# B&R Automation Studio project SceneViewer
Automation Studio 4.7.3.93 SP; technology packages: mappMotion 5.13.1, mappView 5.13.0

## Configuration Config1

CPU PC_any, AutomationRuntime B4.73, Build 4.1.2, Safety 0.0, Vc V4.72.3

### Task classes (Cpu.sw)
```
Cyclic#1 (cycle 1000 us, tolerance 0 us):
  Vis <- Vis.prg
  Trak <- Trak.prg
  SVControl <- SVControl.prg
DataObjects: McAcpSys
Binaries: FWRules, McAcpSim, arcoal, arsvcreg, TCData, McAcpDrv, arflatprv, udbdef, mvLoader, iomap, Config_1, arconfig, asfw, ashwac, sysconf, User, Role, ashwd, Config_3
Libraries: BeEasyTrak, SceneView, McBase, McAxis, McAcpTrak, standard, AsBrStr, AsMath, MpAxis, MpBase, McAcpAx, runtime, astime, fileio, powerlnk, asieccon, arssl
```

### Hardware
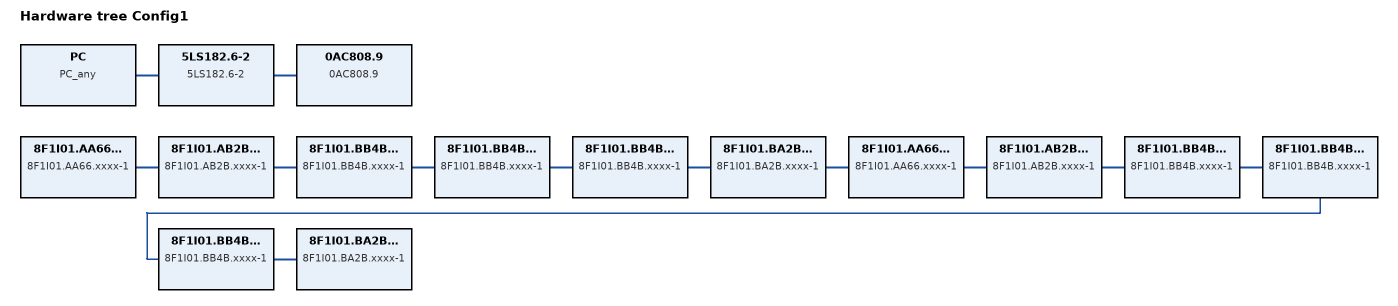
```
0AC808.9 : 0AC808.9 v1.0.0.0  [ETH1 -> 5LS182.6-2.IF1 [Cable Type=PowerlinkCable, Length=10, Version=1.0.0.2]; ETH2 -> 8F1I01.AA66.xxxx-1.PLK3 [Cable Type=PowerlinkCable, Length=10, Version=1.0.0.2]]
5LS182.6-2 : 5LS182.6-2 v1.7.0.0  [SL -> PC.SL1]
8F1I01.AA66.xxxx-1 : 8F1I01.AA66.xxxx-1 v1.0.0.2  [PLK2 -> 8F1I01.AB2B.xxxx-1.PLK1 [Cable Type=PowerlinkCable, Length=10, Version=1.0.0.2]; PLK3 -> 0AC808.9.ETH2 [Cable Type=PowerlinkCable, Length=10, Version=1.0.0.2]]
  DriveConfiguration:
    McTypeID = LLMConfig
  DriveConfiguration/Segment:
    Shape = STRAIGHT660
    SegmentReference = gSeg_Main_1
    StopReaction = UseAssemblySetting
    SpeedFilter = UseAssemblySetting
8F1I01.AA66.xxxx-1a : 8F1I01.AA66.xxxx-1 v1.0.0.2  [PLK1 -> 8F1I01.BA2B.xxxx-1a.PLK2 [Cable Type=PowerlinkCable, Length=10, Version=1.0.0.2]; PLK2 -> 8F1I01.AB2B.xxxx-1a.PLK1 [Cable Type=PowerlinkCable, Length=10, Version=1.0.0.2]]
  DriveConfiguration:
    McTypeID = LLMConfig
  DriveConfiguration/Segment:
    Shape = STRAIGHT660
    SegmentReference = gSeg_Main_7
    StopReaction = UseAssemblySetting
    SpeedFilter = UseAssemblySetting
8F1I01.AB2B.xxxx-1 : 8F1I01.AB2B.xxxx-1 v1.0.0.2  [PLK1 -> 8F1I01.AA66.xxxx-1.PLK2 [Cable Type=PowerlinkCable, Length=10, Version=1.0.0.2]; PLK2 -> 8F1I01.BB4B.xxxx-1.PLK1 [Cable Type=PowerlinkCable, Length=10, Version=1.0.0.2]]
  DriveConfiguration:
    McTypeID = LLMConfig
  DriveConfiguration/Segment:
    Shape = STRAIGHT105_TO_CIRCULAR
    SegmentReference = gSeg_Main_2
    StopReaction = UseAssemblySetting
    SpeedFilter = UseAssemblySetting
8F1I01.AB2B.xxxx-1a : 8F1I01.AB2B.xxxx-1 v1.0.0.2  [PLK1 -> 8F1I01.AA66.xxxx-1a.PLK2 [Cable Type=PowerlinkCable, Length=10, Version=1.0.0.2]; PLK2 -> 8F1I01.BB4B.xxxx-1c.PLK1 [Cable Type=PowerlinkCable, Length=10, Version=1.0.0.2]]
  DriveConfiguration:
    McTypeID = LLMConfig
  DriveConfiguration/Segment:
    Shape = STRAIGHT105_TO_CIRCULAR
    SegmentReference = gSeg_Main_8
    StopReaction = UseAssemblySetting
    SpeedFilter = UseAssemblySetting
8F1I01.BA2B.xxxx-1 : 8F1I01.BA2B.xxxx-1 v1.0.0.2  [PLK1 -> 8F1I01.BB4B.xxxx-1e.PLK2 [Cable Type=PowerlinkCable, Length=10, Version=1.0.0.2]]
  DriveConfiguration:
    McTypeID = LLMConfig
  DriveConfiguration/Segment:
    Shape = CIRCULAR_TO_STRAIGHT105
    SegmentReference = gSeg_Main_12
    StopReaction = UseAssemblySetting
    SpeedFilter = UseAssemblySetting
8F1I01.BA2B.xxxx-1a : 8F1I01.BA2B.xxxx-1 v1.0.0.2  [PLK1 -> 8F1I01.BB4B.xxxx-1b.PLK2 [Cable Type=PowerlinkCable, Length=10, Version=1.0.0.2]; PLK2 -> 8F1I01.AA66.xxxx-1a.PLK1 [Cable Type=PowerlinkCable, Length=10, Version=1.0.0.2]]
  DriveConfiguration:
    McTypeID = LLMConfig
  DriveConfiguration/Segment:
    Shape = CIRCULAR_TO_STRAIGHT105
    SegmentReference = gSeg_Main_6
    StopReaction = UseAssemblySetting
    SpeedFilter = UseAssemblySetting
8F1I01.BB4B.xxxx-1 : 8F1I01.BB4B.xxxx-1 v1.0.0.2  [PLK1 -> 8F1I01.AB2B.xxxx-1.PLK2 [Cable Type=PowerlinkCable, Length=10, Version=1.0.0.2]; PLK2 -> 8F1I01.BB4B.xxxx-1a.PLK1 [Cable Type=PowerlinkCable, Length=10, Version=1.0.0.2]]
  DriveConfiguration:
    McTypeID = LLMConfig
  DriveConfiguration/Segment:
    Shape = CIRCULAR
    SegmentReference = gSeg_Main_3
    StopReaction = UseAssemblySetting
    SpeedFilter = UseAssemblySetting
8F1I01.BB4B.xxxx-1a : 8F1I01.BB4B.xxxx-1 v1.0.0.2  [PLK1 -> 8F1I01.BB4B.xxxx-1.PLK2 [Cable Type=PowerlinkCable, Length=10, Version=1.0.0.2]; PLK2 -> 8F1I01.BB4B.xxxx-1b.PLK1 [Cable Type=PowerlinkCable, Length=10, Version=1.0.0.2]]
  DriveConfiguration:
    McTypeID = LLMConfig
  DriveConfiguration/Segment:
    Shape = CIRCULAR
    SegmentReference = gSeg_Main_4
    StopReaction = UseAssemblySetting
    SpeedFilter = UseAssemblySetting
8F1I01.BB4B.xxxx-1b : 8F1I01.BB4B.xxxx-1 v1.0.0.2  [PLK1 -> 8F1I01.BB4B.xxxx-1a.PLK2 [Cable Type=PowerlinkCable, Length=10, Version=1.0.0.2]; PLK2 -> 8F1I01.BA2B.xxxx-1a.PLK1 [Cable Type=PowerlinkCable, Length=10, Version=1.0.0.2]]
  DriveConfiguration:
    McTypeID = LLMConfig
  DriveConfiguration/Segment:
    Shape = CIRCULAR
    SegmentReference = gSeg_Main_5
    StopReaction = UseAssemblySetting
    SpeedFilter = UseAssemblySetting
8F1I01.BB4B.xxxx-1c : 8F1I01.BB4B.xxxx-1 v1.0.0.2  [PLK1 -> 8F1I01.AB2B.xxxx-1a.PLK2 [Cable Type=PowerlinkCable, Length=10, Version=1.0.0.2]; PLK2 -> 8F1I01.BB4B.xxxx-1d.PLK1 [Cable Type=PowerlinkCable, Length=10, Version=1.0.0.2]]
  DriveConfiguration:
    McTypeID = LLMConfig
  DriveConfiguration/Segment:
    Shape = CIRCULAR
    SegmentReference = gSeg_Main_9
    StopReaction = UseAssemblySetting
    SpeedFilter = UseAssemblySetting
8F1I01.BB4B.xxxx-1d : 8F1I01.BB4B.xxxx-1 v1.0.0.2  [PLK1 -> 8F1I01.BB4B.xxxx-1c.PLK2 [Cable Type=PowerlinkCable, Length=10, Version=1.0.0.2]; PLK2 -> 8F1I01.BB4B.xxxx-1e.PLK1 [Cable Type=PowerlinkCable, Length=10, Version=1.0.0.2]]
  DriveConfiguration:
    McTypeID = LLMConfig
  DriveConfiguration/Segment:
    Shape = CIRCULAR
    SegmentReference = gSeg_Main_10
    StopReaction = UseAssemblySetting
    SpeedFilter = UseAssemblySetting
8F1I01.BB4B.xxxx-1e : 8F1I01.BB4B.xxxx-1 v1.0.0.2  [PLK1 -> 8F1I01.BB4B.xxxx-1d.PLK2 [Cable Type=PowerlinkCable, Length=10, Version=1.0.0.2]; PLK2 -> 8F1I01.BA2B.xxxx-1.PLK1 [Cable Type=PowerlinkCable, Length=10, Version=1.0.0.2]]
  DriveConfiguration:
    McTypeID = LLMConfig
  DriveConfiguration/Segment:
    Shape = CIRCULAR
    SegmentReference = gSeg_Main_11
    StopReaction = UseAssemblySetting
    SpeedFilter = UseAssemblySetting
PC : PC_any v1.1.0.0 (OrderNumber=PC)
  ConfigurationID = SceneViewer_Config1
  SystemTick = 1000
  Cyclic1Duration = 1000
  Cyclic1Tolerance = 0
  Cyclic2Duration = 2000
  FileDevice1
  FileDeviceName1 = SvgData
  FileDevicePath1 = C:\Trak\Scene
  ActivateOpcUa = 1
  OpcUaInformationModels_PV_Version = 1
```

### Config_1.assembly - PC/mappMotion/Config_1.assembly
```
Element gAssembly_1 (Type=assembly)
  Tracks:
    TrackSeparation = 0.030
    Track[1]:
      Segments:
        SegmentRef[1] = ::gSeg_Main_1
        SegmentRef[2] = ::gSeg_Main_2
        SegmentRef[3] = ::gSeg_Main_3
        SegmentRef[4] = ::gSeg_Main_4
        SegmentRef[5] = ::gSeg_Main_5
        SegmentRef[6] = ::gSeg_Main_6
        SegmentRef[7] = ::gSeg_Main_7
        SegmentRef[8] = ::gSeg_Main_8
        SegmentRef[9] = ::gSeg_Main_9
        SegmentRef[10] = ::gSeg_Main_10
        SegmentRef[11] = ::gSeg_Main_11
        SegmentRef[12] = ::gSeg_Main_12
      Position = Absolute
        SegmentCountDirection = RightToLeft
        Translation:
          X = 0.0
          Y = 0.0
          Z = 0.0
        Orientation:
          Angle1 = 0.0
          Angle2 = 0.0
          Angle3 = 0.0
  CommonSegmentSettings:
    SegmentSimulationOnPLC = Off
    StopReaction = InductionHalt
    SpeedFilter = NotUsed
    ControllerParameters:
      DefaultParameter:
        Controller:
          Position:
            ProportionalGain = 0.0
          Speed:
            ProportionalGain = 0.0
            IntegrationTime = 0.0
          FeedForward:
            TotalMass = 0.0
            ForcePositive = 0.0
            ForceNegative = 0.0
            SpeedForceFactor = 0.0
            ForceLoad = 0.0
        MovementErrorLimits:
          PositionError = 0.0
          VelocityError = 0.0
      AdditionalParameterSets = NotUsed
    ScopeOfErrorReaction = Assembly
    ShuttleIdentificationTime = 0
  Shuttles:
    MaxShuttleCount = 10
    DistanceReserve:
      Collision = 0.002
      ErrorStop = 0.006
    ShuttleStereotypes:
      ShuttleStRef[1] = ShuttleStereotype_1
    MagnetPlateConfigurations:
      ShuttleType[1] = 8F1SA.100.xxxxxx-x
    CollisionAvoidance:
      Strategy = Constant
      MaximumModelDimensions:
        Length:
          ExtentToFront = 0.025
          ExtentToBack = 0.025
        Width:
          Width = 0.046
  AssemblyFeatures:
    AssemblyFeatureRef[1] = AssemblyFeature_1
  Visualization:
    MonitoringPv = ::gShuttleMon
    ProcessingTaskClass = 2
```

### Config_2.sector - PC/mappMotion/Config_2.sector
```
Element Sector_1 (Type=sector)
  Type = Composed
    StartSegment:
      SegmentRef = ::gSeg_Main_1
    IntermediateSegments:
      SegmentRef[1] = ::gSeg_Main_2
      SegmentRef[2] = ::gSeg_Main_3
      SegmentRef[3] = ::gSeg_Main_4
      SegmentRef[4] = ::gSeg_Main_5
      SegmentRef[5] = ::gSeg_Main_6
      SegmentRef[6] = ::gSeg_Main_7
      SegmentRef[7] = ::gSeg_Main_8
      SegmentRef[8] = ::gSeg_Main_9
      SegmentRef[9] = ::gSeg_Main_10
      SegmentRef[10] = ::gSeg_Main_11
    EndSegment:
      SegmentRef = ::gSeg_Main_12
      PositionRelativeTo = FromEnd
```

### Config_3.shuttlestereotype - PC/mappMotion/Config_3.shuttlestereotype
```
Element ShuttleStereotype_1 (Type=shuttlestereotype)
  MeasurementUnit = 5067858
  MeasurementResolution = 0.00001
  MovementLimits = Internal
    VelocityIsReadOnly = 0
    Velocity:
      Velocity = 4.0
    AccelerationIsReadOnly = 0
    Acceleration:
      Acceleration = 20
    DecelerationIsReadOnly = 0
    Deceleration:
      Deceleration = 20
  JerkFilter = Used
    JerkTime = 0.02
  UserData:
    Size = 0
```

### Config_4.assemblyfeature - PC/mappMotion/Config_4.assemblyfeature
```
Element AssemblyFeature_1 (Type=assemblyfeature)
  Type = InitShuttleSim
    InitShuttleSim[1]:
      SectorRef = Sector_1
      Orientation = Positive
      ShuttleDefinition = ShuttleSetDefinition
        StartPosition = 0.0
        NumberOfShuttles = 5
        DistnaceBetweenShuttles = 0.2
```

### cfgSV.mprecipexml - PC/mappServices/cfgSV.mprecipexml
```
Element gRecipeScnViewer (Type=mprecipexml)
```

## Logical view

Binary libraries used (declarations not repeated): operator, runtime, astime, AsIecCon, McBase 5.13.1, McAxis 5.13.1, McAcpTrak 5.13.1, standard, AsBrStr, AsMath, MpAxis 5.13.1, MpBase 5.13.0, McAcpAx 5.13.1

### Segments.var
```iecst
VAR
	gSeg_Main_1 : McSegmentType;
	gSeg_Main_2 : McSegmentType;
	gSeg_Main_3 : McSegmentType;
	gSeg_Main_4 : McSegmentType;
	gSeg_Main_5 : McSegmentType;
	gSeg_Main_6 : McSegmentType;
	gSeg_Main_7 : McSegmentType;
	gSeg_Main_8 : McSegmentType;
	gSeg_Main_9 : McSegmentType;
	gSeg_Main_10 : McSegmentType;
	gSeg_Main_11 : McSegmentType;
	gSeg_Main_12 : McSegmentType;
END_VAR
```

### Package Logical/Libraries - Global libraries

### Library Logical/Libraries/BeEasyTrak (IEC)

#### Types.typ - Exported data types
```iecst
TYPE
	Barrier_typ : 	STRUCT
		BarrierReadInfo : MC_BR_BarrierReadInfo_AcpTrak;
		BarrierCommand : MC_BR_BarrierCommand_AcpTrak;
	END_STRUCT;
	TrgPoint_typ : 	STRUCT
		TrgPointGetInfo : MC_BR_TrgPointGetInfo_AcpTrak;
		TrgPointEnable : MC_BR_TrgPointEnable_AcpTrak;
	END_STRUCT;
	ShuttleUserData_typ : 	STRUCT
		Color : Color_enum;
	END_STRUCT;
	Color_enum :
		(
		GRAY := 0,
		GREEN := 1,
		BLUE := 2,
		RED := 3,
		ORANGE := 4,
		YELLOW,
		WHITE
		);
END_TYPE
```

#### Constants.var - Exported constants
```iecst
VAR CONSTANT
	MAX_SHUTTLES : UINT := 5;
	NUM_SHUTTLES : UINT := 5;
END_VAR
```

#### BeEasyTrak.fun - Exported functions and function blocks
```iecst
{REDUND_ERROR} FUNCTION_BLOCK BE_TrgPoint (*TODO: Add your comment here*) (*$GROUP=User,$CAT=User,$GROUPICON=User.png,$CATICON=User.png*)
	VAR_INPUT
		ProcessPoint : REFERENCE TO McProcessPointType;
		Enable : BOOL;
	END_VAR
	VAR_OUTPUT
		ShuttleAxis : McAxisType;
		Triggered : BOOL;
	END_VAR
	VAR
		State : USINT;
		TrgPoint : TrgPoint_typ;
	END_VAR
END_FUNCTION_BLOCK

{REDUND_ERROR} FUNCTION_BLOCK BE_SimStartup (*TODO: Add your comment here*) (*$GROUP=User,$CAT=User,$GROUPICON=User.png,$CATICON=User.png*)
	VAR_INPUT
		Assembly : REFERENCE TO McAssemblyType;
		Sector : REFERENCE TO McSectorType;
		Execute : BOOL;
	END_VAR
	VAR_OUTPUT
		ShuttleAxisArray : ARRAY[1..MAX_SHUTTLES] OF McAxisType;
		Done : BOOL;
	END_VAR
	VAR
		AsmReadInfo : MC_BR_AsmReadInfo_AcpTrak;
		AddShuttle : MC_BR_SecAddShuttle_AcpTrak;
		ElasticMoveVel : MC_BR_ElasticMoveVel_AcpTrak;
		State : USINT;
		i : USINT := 1;
		zzEdge00000 : BOOL;
	END_VAR
END_FUNCTION_BLOCK

{REDUND_ERROR} FUNCTION_BLOCK BE_Rate (*TODO: Add your comment here*) (*$GROUP=User,$CAT=User,$GROUPICON=User.png,$CATICON=User.png*)
	VAR_INPUT
		ProcessPoint : REFERENCE TO McProcessPointType;
		Enable : BOOL;
	END_VAR
	VAR_OUTPUT
		PPM : UINT;
		PPM_Instant : REAL;
		PPH : UINT;
		PPH_Instant : REAL;
	END_VAR
	VAR
		Counter : UINT;
		State : USINT;
		TrgPoint : BE_TrgPoint;
		TON_InstantRate : TON;
		TON_PPM : TON;
	END_VAR
END_FUNCTION_BLOCK

{REDUND_ERROR} FUNCTION_BLOCK BE_FindShuttles (*TODO: Add your comment here*) (*$GROUP=User,$CAT=User,$GROUPICON=User.png,$CATICON=User.png*)
	VAR_INPUT
		Assembly : REFERENCE TO USINT;
		Execute : {REDUND_UNREPLICABLE} BOOL;
	END_VAR
	VAR_OUTPUT
		NumShuttlesFound : UINT;
		ShuttleAxisArray : ARRAY[1..MAX_SHUTTLES] OF McAxisType;
		Done : {REDUND_UNREPLICABLE} BOOL;
		Error : BOOL;
		Busy : BOOL;
	END_VAR
	VAR
		i : USINT;
		AsmGetShuttle : MC_BR_AsmGetShuttle_AcpTrak;
		State : USINT;
	END_VAR
END_FUNCTION_BLOCK

{REDUND_ERROR} FUNCTION_BLOCK BE_MoveOnSector (*TODO: Add your comment here*) (*$GROUP=User,$CAT=User,$GROUPICON=User.png,$CATICON=User.png*)
	VAR_INPUT
		Execute : {REDUND_UNREPLICABLE} BOOL;
		Sector : REFERENCE TO McSectorType;
		Velocity : REAL;
		Acceleration : REAL;
		Deceleration : REAL;
		AxisArray : ARRAY[1..MAX_SHUTTLES] OF McAxisType;
		Assembly : REFERENCE TO McAssemblyType;
	END_VAR
	VAR_OUTPUT
		NumShuttles : UINT;
		Done : {REDUND_UNREPLICABLE} BOOL;
	END_VAR
	VAR
		RoutedMoveVel : MC_BR_RoutedMoveVel_AcpTrak;
		AsmGetShuttle : MC_BR_AsmGetShuttle_AcpTrak;
		i : UINT;
		State : USINT;
		zzEdge00000 : BOOL;
	END_VAR
END_FUNCTION_BLOCK

{REDUND_ERROR} FUNCTION_BLOCK BE_AsmStop (*TODO: Add your comment here*) (*$GROUP=User,$CAT=User,$GROUPICON=User.png,$CATICON=User.png*)
	VAR_INPUT
		Execute : {REDUND_UNREPLICABLE} BOOL;
		AxisArray : {REDUND_UNREPLICABLE} ARRAY[1..MAX_SHUTTLES] OF McAxisType;
		Deceleration : REAL;
		NumShuttles : UINT;
	END_VAR
	VAR_OUTPUT
		Done : {REDUND_UNREPLICABLE} BOOL;
	END_VAR
	VAR
		State : USINT;
		Stop : MC_Stop;
		i : UINT;
	END_VAR
END_FUNCTION_BLOCK
```

#### BE_TrgPoint.st
```iecst
(* TODO: Add your comment here *)
FUNCTION_BLOCK BE_TrgPoint

	TrgPoint.TrgPointEnable.ProcessPoint := ADR(ProcessPoint);
	TrgPoint.TrgPointGetInfo.ProcessPoint := ADR(ProcessPoint);

	TrgPoint.TrgPointEnable.Enable := Enable;

	CASE State OF
		0:
			IF TrgPoint.TrgPointEnable.EventCount > 0 THEN
				TrgPoint.TrgPointGetInfo.Execute := TRUE;
			END_IF

			IF TrgPoint.TrgPointGetInfo.TrgPointInfo.Event = mcACPTRAK_TP_PASSED_POSITIVE THEN
				ShuttleAxis := TrgPoint.TrgPointGetInfo.TrgPointInfo.Axis;
				TrgPoint.TrgPointGetInfo.Execute := FALSE;
				Triggered := TRUE;
				State := 1;
			END_IF

		1:
			Triggered := FALSE;
			State := 0;

	END_CASE

	TrgPoint.TrgPointEnable();
	TrgPoint.TrgPointGetInfo();

END_FUNCTION_BLOCK
```

#### BE_SimStartup.st
```iecst
(* TODO: Add your comment here *)
FUNCTION_BLOCK BE_SimStartup

	AsmReadInfo.Assembly := ADR(Assembly);
	AsmReadInfo.Enable := TRUE;

	CASE State OF
		0: //POWER_ON
			IF Execute THEN
				State := 1;
			END_IF

		1: //ADD_SHUTTLES
			AddShuttle.Sector := ADR(Sector);
			AddShuttle.Position := (i - 1) * 0.1;
			AddShuttle.Execute := TRUE;

			IF AddShuttle.Done  THEN
				ShuttleAxisArray[i] := AddShuttle.Axis;
				AddShuttle.Execute := FALSE;
				i := i + 1;
			END_IF

			IF i > NUM_SHUTTLES THEN
				i := 1;
				State := 2;
			END_IF

		2: //MOVE_SHUTTLES

			IF EDGEPOS(ElasticMoveVel.Active) THEN
				i := i + 1;
			ELSIF ShuttleAxisArray[i].controlif <> 0 THEN
				ElasticMoveVel.Axis := ADR(ShuttleAxisArray[i]);
				ElasticMoveVel.Velocity := 2;
				ElasticMoveVel.Acceleration := 10;
				ElasticMoveVel.Deceleration := 10;
				ElasticMoveVel.Execute := TRUE;
			END_IF

			IF i > NUM_SHUTTLES THEN
				State := 3;
			END_IF
//
		3: //STANDBY
			Done := TRUE;
			IF NOT Execute THEN
				Done := FALSE;
				State := 0;
			END_IF

	END_CASE

	AddShuttle();
	AsmReadInfo();
	ElasticMoveVel();
	ElasticMoveVel.Execute := FALSE;

END_FUNCTION_BLOCK
```

#### BE_Rate.st
```iecst
(* TODO: Add your comment here *)
FUNCTION_BLOCK BE_Rate

	CASE State OF
		0:
			IF Enable THEN
				State := 1;
			END_IF

		1:
			TON_InstantRate.PT := T#60m;
			TON_InstantRate.IN := TRUE;

			TrgPoint.ProcessPoint := ADR(ProcessPoint);
			TrgPoint.Enable := TRUE;

			IF TrgPoint.Triggered THEN
				Counter := Counter + 1;

				TON_InstantRate.IN := FALSE;
				IF TIME_TO_REAL(TON_InstantRate.ET) <> 0 THEN
					PPM_Instant := 1000 / TIME_TO_REAL(TON_InstantRate.ET);
					PPH_Instant := 60 * 1000 / TIME_TO_REAL(TON_InstantRate.ET);
				END_IF
			END_IF

			TON_PPM.PT := T#60s;
			TON_PPM.IN := TRUE;

			IF TON_PPM.Q THEN
				TON_PPM.IN := FALSE;
				PPM := Counter;
				Counter := 0;
			END_IF

			PPH := PPM * 60;

	END_CASE

	TON_InstantRate;
	TrgPoint();
	TON_PPM();

END_FUNCTION_BLOCK
```

#### BE_FindShuttles.st
```iecst
(* TODO: Add your comment here *)
FUNCTION_BLOCK BE_FindShuttles
	AsmGetShuttle.Assembly := ADR(Assembly);

	IF AsmGetShuttle.Error THEN
		Error := TRUE;
		State := 4;
	END_IF

	CASE State OF
		0:
			IF Execute THEN
				i := 1;
				Busy := TRUE;
				State := 1;
			END_IF

		1:
			AsmGetShuttle.Enable := TRUE;
			IF AsmGetShuttle.Valid THEN
				NumShuttlesFound := AsmGetShuttle.TotalCount;
				IF AsmGetShuttle.Axis.controlif <> 0 THEN
					ShuttleAxisArray[i] := AsmGetShuttle.Axis;
				END_IF
				IF AsmGetShuttle.RemainingCount > 0 THEN
					AsmGetShuttle.Next := TRUE;
					State := 2;
				ELSE
					State := 3;
				END_IF
			END_IF

		2:
			AsmGetShuttle.Next := FALSE;
			i := i + 1;
			State := 1;

		3:
			Done := TRUE;
			IF NOT Execute THEN
				brsmemset(ADR(ShuttleAxisArray),0,SIZEOF(ShuttleAxisArray));
				AsmGetShuttle.Enable := FALSE;
				NumShuttlesFound := 0;
				Done := FALSE;
				Busy := FALSE;
				State := 0;
			END_IF

		4: //error state

	END_CASE

	AsmGetShuttle();

END_FUNCTION_BLOCK
```

#### BE_MoveOnSector.st
```iecst
(* TODO: Add your comment here *)
FUNCTION_BLOCK BE_MoveOnSector
	CASE State OF
		0:
			IF Execute THEN
				i := 1;
				State := 1;
			END_IF

		1:
			AsmGetShuttle.Assembly := ADR(Assembly);
			AsmGetShuttle.Enable := TRUE;
			IF AsmGetShuttle.Valid THEN
				NumShuttles := AsmGetShuttle.TotalCount;
				AsmGetShuttle.Enable := FALSE;
				State := 2;
			END_IF

		2:
			IF EDGEPOS(RoutedMoveVel.Active) THEN
				i := i + 1;
			ELSIF AxisArray[i].controlif <> 0 THEN
				RoutedMoveVel.Sector := ADR(Sector);
				RoutedMoveVel.Axis := ADR(AxisArray[i]);
				RoutedMoveVel.Position := 0;
				RoutedMoveVel.RouteVelocity := Velocity;
				RoutedMoveVel.Velocity := Velocity;
				RoutedMoveVel.Acceleration := Acceleration;
				RoutedMoveVel.Deceleration := Deceleration;
				RoutedMoveVel.Execute := TRUE;
			END_IF

			IF i > NumShuttles THEN
				State := 3;
			END_IF

		3:
			Done := TRUE;
			State := 4;

		4:
			IF NOT Execute THEN
				Done := FALSE;
				NumShuttles := 0;
				State := 0;
			END_IF

	END_CASE

	AsmGetShuttle();
	RoutedMoveVel();
	RoutedMoveVel.Execute := FALSE;

END_FUNCTION_BLOCK
```

#### BE_AsmStop.st
```iecst
(* TODO: Add your comment here *)
FUNCTION_BLOCK BE_AsmStop
	CASE State OF
		0:
			IF Execute THEN
				i := 1;
				State := 1;
			END_IF

		1:

			Stop.Deceleration := Deceleration;
			Stop.Axis := ADR(AxisArray[i]);
			Stop.Execute := TRUE;

			IF i >= NumShuttles THEN
				Done := TRUE;
				State := 3;
			ELSE
				State := 2;
			END_IF

		2:
			Stop.Execute := FALSE;
			i := i + 1;
			State := 1;

		3:
			IF NOT Execute THEN
				State := 0;
				Done := FALSE;
				Stop.Execute := FALSE;
			END_IF

	END_CASE

	Stop();

END_FUNCTION_BLOCK
```

### Library Logical/Libraries/SceneView (IEC)

#### Types.typ - Exported data types
```iecst
TYPE
	SceneViewCoord_typ : 	STRUCT
		X : REAL;
		Y : REAL;
		Z : REAL;
	END_STRUCT;
	SceneViewCamera_typ : 	STRUCT
		Perspective : BOOL;
		Zoom : REAL;
		Fov : REAL;
		ViewPoint : SceneViewCoord_typ;
		ViewVector : SceneViewCoord_typ;
		OrientationVector : SceneViewCoord_typ;
	END_STRUCT;
END_TYPE
```

#### Constants.var - Exported constants
```iecst
VAR CONSTANT
	PI : REAL := 3.14159265359;
END_VAR
```

#### SceneView.fun - Exported functions and function blocks
```iecst
{REDUND_ERROR} FUNCTION_BLOCK SV_BE_MoveView (*TODO: Add your comment here*) (*$GROUP=User,$CAT=User,$GROUPICON=User.png,$CATICON=User.png*)
	VAR_INPUT
		Execute : BOOL;
		PointA : SceneViewCamera_typ;
		PointB : SceneViewCamera_typ;
		TravelTime : TIME;
	END_VAR
	VAR_OUTPUT
		Error : BOOL;
		Done : BOOL;
		SceneViewPos : SceneViewCamera_typ;
	END_VAR
	VAR
		TON_ViewChange : TON;
		State : USINT;
		ChangeRate : SceneViewCamera_typ;
	END_VAR
END_FUNCTION_BLOCK

{REDUND_ERROR} FUNCTION_BLOCK SV_BE_FocalPointMove (*TODO: Add your comment here*) (*$GROUP=User,$CAT=User,$GROUPICON=User.png,$CATICON=User.png*)
	VAR_INPUT
		FocalPointA : SceneViewCoord_typ;
		FocalPointB : SceneViewCoord_typ;
		Execute : BOOL;
		PointA : SceneViewCamera_typ;
		PointB : SceneViewCamera_typ;
		TravelTime : TIME;
	END_VAR
	VAR_OUTPUT
		Error : BOOL;
		Done : BOOL;
		FocalPointPos : SceneViewCoord_typ;
		SceneViewPos : SceneViewCamera_typ;
	END_VAR
	VAR
		TON_ViewChange : TON;
		State : USINT;
		FocalPointChangeRate : SceneViewCoord_typ;
		ChangeRate : SceneViewCamera_typ;
	END_VAR
END_FUNCTION_BLOCK

{REDUND_ERROR} FUNCTION_BLOCK SV_BE_RadialMove
	VAR_INPUT
		FocalPointA : SceneViewCoord_typ;
		FocalPointB : SceneViewCoord_typ;
		Execute : BOOL;
		PointA : SceneViewCamera_typ;
		PointB : SceneViewCamera_typ;
		TravelTime : TIME;
	END_VAR
	VAR_OUTPUT
		Error : BOOL;
		Done : BOOL;
		FocalPointPos : SceneViewCoord_typ;
		SceneViewPos : SceneViewCamera_typ;
	END_VAR
	VAR
		FocalPointChangeRate : SceneViewCoord_typ;
		TON_ViewChange : TON;
		State : USINT;
		ChangeRate : SceneViewCamera_typ;
		RadiusA : REAL;
		RadiusB : REAL;
		RadiusChangeRate : REAL;
		OutputRadius : REAL;
		AngleA : REAL;
		AngleB : REAL;
		AngleChangeRate : REAL;
		OutputAngle : REAL;
	END_VAR
END_FUNCTION_BLOCK
```

#### SV_BE_MoveView.st
```iecst
(* TODO: Add your comment here *)
FUNCTION_BLOCK SV_BE_MoveView
	IF Error THEN
		State := 50;
	ELSIF NOT Execute THEN
		State := 0;
	END_IF

	CASE State OF
		0:
			Done := FALSE;
			TON_ViewChange.IN := FALSE;

			IF Execute THEN
				IF TIME_TO_REAL(TravelTime) = 0 THEN
					Error := TRUE;
				ELSE
					SceneViewPos := PointA;
					State := 1;
				END_IF
			END_IF

		1:
			ChangeRate.Zoom := (PointB.Zoom - PointA.Zoom) / TIME_TO_REAL(TravelTime);
			ChangeRate.ViewPoint.X := (PointB.ViewPoint.X - PointA.ViewPoint.X) / TIME_TO_REAL(TravelTime);
			ChangeRate.ViewPoint.Y := (PointB.ViewPoint.Y - PointA.ViewPoint.Y) / TIME_TO_REAL(TravelTime);
			ChangeRate.ViewPoint.Z := (PointB.ViewPoint.Z - PointA.ViewPoint.Z) / TIME_TO_REAL(TravelTime);
			ChangeRate.ViewVector.X := (PointB.ViewVector.X - PointA.ViewVector.X) / TIME_TO_REAL(TravelTime);
			ChangeRate.ViewVector.Y := (PointB.ViewVector.Y - PointA.ViewVector.Y) / TIME_TO_REAL(TravelTime);
			ChangeRate.ViewVector.Z := (PointB.ViewVector.Z - PointA.ViewVector.Z) / TIME_TO_REAL(TravelTime);
			ChangeRate.OrientationVector.X := (PointB.OrientationVector.X - PointA.OrientationVector.X) / TIME_TO_REAL(TravelTime);
			ChangeRate.OrientationVector.Y := (PointB.OrientationVector.Y - PointA.OrientationVector.Y) / TIME_TO_REAL(TravelTime);
			ChangeRate.OrientationVector.Z := (PointB.OrientationVector.Z - PointA.OrientationVector.Z) / TIME_TO_REAL(TravelTime);

			State := 2;

		2:
			TON_ViewChange.PT := TravelTime;
			TON_ViewChange.IN := TRUE;
			IF TON_ViewChange.Q THEN
				TON_ViewChange.IN := FALSE;
				State := 3;
			END_IF

			SceneViewPos.Zoom := PointA.Zoom + ChangeRate.Zoom * TIME_TO_REAL(TON_ViewChange.ET);
			SceneViewPos.ViewPoint.X := PointA.ViewPoint.X + ChangeRate.ViewPoint.X * TIME_TO_REAL(TON_ViewChange.ET);
			SceneViewPos.ViewPoint.Y := PointA.ViewPoint.Y + ChangeRate.ViewPoint.Y * TIME_TO_REAL(TON_ViewChange.ET);
			SceneViewPos.ViewPoint.Z := PointA.ViewPoint.Z + ChangeRate.ViewPoint.Z * TIME_TO_REAL(TON_ViewChange.ET);
			SceneViewPos.ViewVector.X := PointA.ViewVector.X + ChangeRate.ViewVector.X * TIME_TO_REAL(TON_ViewChange.ET);
			SceneViewPos.ViewVector.Y := PointA.ViewVector.Y + ChangeRate.ViewVector.Y * TIME_TO_REAL(TON_ViewChange.ET);
			SceneViewPos.ViewVector.Z := PointA.ViewVector.Z + ChangeRate.ViewVector.Z * TIME_TO_REAL(TON_ViewChange.ET);
			SceneViewPos.OrientationVector.X := PointA.OrientationVector.X + ChangeRate.OrientationVector.X * TIME_TO_REAL(TON_ViewChange.ET);
			SceneViewPos.OrientationVector.Y := PointA.OrientationVector.Y + ChangeRate.OrientationVector.Y * TIME_TO_REAL(TON_ViewChange.ET);
			SceneViewPos.OrientationVector.Z := PointA.OrientationVector.Z + ChangeRate.OrientationVector.Z * TIME_TO_REAL(TON_ViewChange.ET);

		3:
			Done := TRUE;

		50:
			IF NOT Execute THEN
				Error := FALSE;
				State := 0;
			END_IF

	END_CASE

	TON_ViewChange();

END_FUNCTION_BLOCK
```

#### SV_BE_FocalPointMove.st
```iecst
(* TODO: Add your comment here *)
FUNCTION_BLOCK SV_BE_FocalPointMove
	IF Error THEN
		State := 50;
	ELSIF NOT Execute THEN
		State := 0;
	END_IF

	CASE State OF
		0:
			Done := FALSE;
			TON_ViewChange.IN := FALSE;

			IF Execute THEN
				IF TIME_TO_REAL(TravelTime) = 0 THEN
					Error := TRUE;
				ELSE
					SceneViewPos := PointA;
					State := 1;
				END_IF
			END_IF

		1:
			SceneViewPos.Perspective := TRUE;
			ChangeRate.Fov := (PointB.Fov - PointA.Fov) / TIME_TO_REAL(TravelTime);
			ChangeRate.Zoom := (PointB.Zoom - PointA.Zoom) / TIME_TO_REAL(TravelTime);
			ChangeRate.ViewPoint.X := (PointB.ViewPoint.X - PointA.ViewPoint.X) / TIME_TO_REAL(TravelTime);
			ChangeRate.ViewPoint.Y := (PointB.ViewPoint.Y - PointA.ViewPoint.Y) / TIME_TO_REAL(TravelTime);
			ChangeRate.ViewPoint.Z := (PointB.ViewPoint.Z - PointA.ViewPoint.Z) / TIME_TO_REAL(TravelTime);

			FocalPointChangeRate.X := (FocalPointB.X - FocalPointA.X) / TIME_TO_REAL(TravelTime);
			FocalPointChangeRate.Y := (FocalPointB.Y - FocalPointA.Y) / TIME_TO_REAL(TravelTime);
			FocalPointChangeRate.Z := (FocalPointB.Z - FocalPointA.Z) / TIME_TO_REAL(TravelTime);
			ChangeRate.OrientationVector.X := (PointB.OrientationVector.X - PointA.OrientationVector.X) / TIME_TO_REAL(TravelTime);
			ChangeRate.OrientationVector.Y := (PointB.OrientationVector.Y - PointA.OrientationVector.Y) / TIME_TO_REAL(TravelTime);
			ChangeRate.OrientationVector.Z := (PointB.OrientationVector.Z - PointA.OrientationVector.Z) / TIME_TO_REAL(TravelTime);

			State := 2;

		2:
			TON_ViewChange.PT := TravelTime;
			TON_ViewChange.IN := TRUE;
			IF TON_ViewChange.Q THEN
				TON_ViewChange.IN := FALSE;
				State := 3;
			END_IF

			FocalPointPos.X := (FocalPointA.X + FocalPointChangeRate.X * TIME_TO_REAL(TON_ViewChange.ET));
			FocalPointPos.Y := (FocalPointA.Y + FocalPointChangeRate.Y * TIME_TO_REAL(TON_ViewChange.ET));
			FocalPointPos.Z := (FocalPointA.Z + FocalPointChangeRate.Z * TIME_TO_REAL(TON_ViewChange.ET));

			SceneViewPos.OrientationVector.X := PointA.OrientationVector.X + ChangeRate.OrientationVector.X * TIME_TO_REAL(TON_ViewChange.ET);
			SceneViewPos.OrientationVector.Y := PointA.OrientationVector.Y + ChangeRate.OrientationVector.Y * TIME_TO_REAL(TON_ViewChange.ET);
			SceneViewPos.OrientationVector.Z := PointA.OrientationVector.Z + ChangeRate.OrientationVector.Z * TIME_TO_REAL(TON_ViewChange.ET);

			SceneViewPos.Fov := PointA.Fov + ChangeRate.Fov * TIME_TO_REAL(TON_ViewChange.ET);
			SceneViewPos.Zoom := PointA.Zoom + ChangeRate.Zoom * TIME_TO_REAL(TON_ViewChange.ET);
			SceneViewPos.ViewPoint.X := PointA.ViewPoint.X + ChangeRate.ViewPoint.X * TIME_TO_REAL(TON_ViewChange.ET);
			SceneViewPos.ViewPoint.Y := PointA.ViewPoint.Y + ChangeRate.ViewPoint.Y * TIME_TO_REAL(TON_ViewChange.ET);
			SceneViewPos.ViewPoint.Z := PointA.ViewPoint.Z + ChangeRate.ViewPoint.Z * TIME_TO_REAL(TON_ViewChange.ET);
			SceneViewPos.ViewVector.X := (FocalPointPos.X - SceneViewPos.ViewPoint.X) / 1000.0;
			SceneViewPos.ViewVector.Y := (FocalPointPos.Y - SceneViewPos.ViewPoint.Y) / 1000.0;
			SceneViewPos.ViewVector.Z := (FocalPointPos.Z - SceneViewPos.ViewPoint.Z) / 1000.0;

		3:
			Done := TRUE;

		50:
			IF NOT Execute THEN
				Error := FALSE;
				State := 0;
			END_IF

	END_CASE

	TON_ViewChange();

END_FUNCTION_BLOCK
```

#### SV_BE_RadialMove.st
```iecst
(* TODO: Add your comment here *)
FUNCTION_BLOCK SV_BE_RadialMove
	IF Error THEN
		State := 50;
	ELSIF NOT Execute THEN
		State := 0;
	END_IF

	CASE State OF
		0:
			Done := FALSE;
			TON_ViewChange.IN := FALSE;

			IF Execute THEN
				IF (TIME_TO_REAL(TravelTime) = 0) THEN
					Error := TRUE;
				ELSE
					SceneViewPos := PointA;
					State := 1;
				END_IF
			END_IF

		1:

			AngleA := atan2((PointA.ViewPoint.Y - FocalPointA.Y),(PointA.ViewPoint.X - FocalPointA.X));
			AngleB := atan2((PointB.ViewPoint.Y - FocalPointB.Y),(PointB.ViewPoint.X - FocalPointB.X));

			RadiusA := (PointA.ViewPoint.X - FocalPointA.X) / COS(AngleA);
			RadiusB := (PointB.ViewPoint.X - FocalPointB.X) / COS(AngleB);

			SceneViewPos.Perspective := TRUE;

			RadiusChangeRate := (RadiusB - RadiusA) / TIME_TO_REAL(TravelTime);
			AngleChangeRate := (AngleB - AngleA) / TIME_TO_REAL(TravelTime);
			ChangeRate.Fov := (PointB.Fov - PointA.Fov) / TIME_TO_REAL(TravelTime);
			ChangeRate.Zoom := (PointB.Zoom - PointA.Zoom) / TIME_TO_REAL(TravelTime);
			ChangeRate.ViewPoint.X := (PointB.ViewPoint.X - PointA.ViewPoint.X) / TIME_TO_REAL(TravelTime);
			ChangeRate.ViewPoint.Y := (PointB.ViewPoint.Y - PointA.ViewPoint.Y) / TIME_TO_REAL(TravelTime);
			ChangeRate.ViewPoint.Z := (PointB.ViewPoint.Z - PointA.ViewPoint.Z) / TIME_TO_REAL(TravelTime);
			ChangeRate.OrientationVector.X := (PointB.OrientationVector.X - PointA.OrientationVector.X) / TIME_TO_REAL(TravelTime);
			ChangeRate.OrientationVector.Y := (PointB.OrientationVector.Y - PointA.OrientationVector.Y) / TIME_TO_REAL(TravelTime);
			ChangeRate.OrientationVector.Z := (PointB.OrientationVector.Z - PointA.OrientationVector.Z) / TIME_TO_REAL(TravelTime);
			FocalPointChangeRate.X := (FocalPointB.X - FocalPointA.X) / TIME_TO_REAL(TravelTime);
			FocalPointChangeRate.Y := (FocalPointB.Y - FocalPointA.Y) / TIME_TO_REAL(TravelTime);
			FocalPointChangeRate.Z := (FocalPointB.Z - FocalPointA.Z) / TIME_TO_REAL(TravelTime);

			State := 2;

		2:
			TON_ViewChange.PT := TravelTime;
			TON_ViewChange.IN := TRUE;
			IF TON_ViewChange.Q THEN
				TON_ViewChange.IN := FALSE;
				State := 3;
			END_IF

			FocalPointPos.X := (FocalPointA.X + FocalPointChangeRate.X * TIME_TO_REAL(TON_ViewChange.ET));
			FocalPointPos.Y := (FocalPointA.Y + FocalPointChangeRate.Y * TIME_TO_REAL(TON_ViewChange.ET));
			FocalPointPos.Z := (FocalPointA.Z + FocalPointChangeRate.Z * TIME_TO_REAL(TON_ViewChange.ET));

			OutputAngle := AngleA + AngleChangeRate * TIME_TO_REAL(TON_ViewChange.ET);
			OutputRadius := RadiusA + RadiusChangeRate * TIME_TO_REAL(TON_ViewChange.ET);

			SceneViewPos.ViewPoint.X := (OutputRadius * COS(OutputAngle)) + FocalPointPos.X;
			SceneViewPos.ViewPoint.Y := (OutputRadius * SIN(OutputAngle)) + FocalPointPos.Y;

			SceneViewPos.Fov := PointA.Fov + ChangeRate.Fov * TIME_TO_REAL(TON_ViewChange.ET);
			SceneViewPos.Zoom := PointA.Zoom + ChangeRate.Zoom * TIME_TO_REAL(TON_ViewChange.ET);
			SceneViewPos.ViewPoint.Z := PointA.ViewPoint.Z + ChangeRate.ViewPoint.Z * TIME_TO_REAL(TON_ViewChange.ET);
			SceneViewPos.ViewVector.X := (FocalPointPos.X - SceneViewPos.ViewPoint.X) / 1000.0;
			SceneViewPos.ViewVector.Y := (FocalPointPos.Y - SceneViewPos.ViewPoint.Y) / 1000.0;
			SceneViewPos.ViewVector.Z := (FocalPointPos.Z - SceneViewPos.ViewPoint.Z) / 1000.0;
			SceneViewPos.OrientationVector.X := PointA.OrientationVector.X + ChangeRate.OrientationVector.X * TIME_TO_REAL(TON_ViewChange.ET);
			SceneViewPos.OrientationVector.Y := PointA.OrientationVector.Y + ChangeRate.OrientationVector.Y * TIME_TO_REAL(TON_ViewChange.ET);
			SceneViewPos.OrientationVector.Z := PointA.OrientationVector.Z + ChangeRate.OrientationVector.Z * TIME_TO_REAL(TON_ViewChange.ET);

		3:
			Done := TRUE;

		50:
			IF NOT Execute THEN
				Error := FALSE;
				State := 0;
			END_IF

	END_CASE

	TON_ViewChange();

END_FUNCTION_BLOCK
```

### Program Logical/Vis (IEC)

#### Variables.var
```iecst
VAR
	Vis : McAcpTrakAssemblyVisData;
	SizeofVis : UDINT;
	NumVisShuttle : USINT;
	i : USINT;
	pUserData : REFERENCE TO ShuttleUserData_typ;
	SizeofUserData : UDINT;
END_VAR
```

#### Main.st
```iecst
PROGRAM _INIT
    // size of Vis structure - this value has to be entered in B&R scene viewer (PVI -> Options -> Size)
	SizeofVis := SIZEOF(Vis);
	// max number of displayed shuttles
	NumVisShuttle := SIZEOF(Vis.Shuttle) / SIZEOF(Vis.Shuttle[0]);

	SizeofUserData := SIZEOF(pUserData);
END_PROGRAM

PROGRAM _CYCLIC
	FOR i:=0 TO (NumVisShuttle-1) DO
		IF gShuttleMon.Shuttle[i].Available THEN
			// format selected monitor data to fit B&R scene viewer
			Vis.Shuttle[i].Available    := 1;
			Vis.Shuttle[i].PositionX    := LREAL_TO_REAL(gShuttleMon.Shuttle[i].Position.X);
			Vis.Shuttle[i].PositionY    := LREAL_TO_REAL(gShuttleMon.Shuttle[i].Position.Y);
			Vis.Shuttle[i].RotationZ    := LREAL_TO_REAL(gShuttleMon.Shuttle[i].Orientation.Angle1);
			Vis.Shuttle[i].ExtentToFront    := LREAL_TO_REAL(gShuttleMon.Shuttle[i].ExtentToFront);
			Vis.Shuttle[i].ExtentToBack        := LREAL_TO_REAL(gShuttleMon.Shuttle[i].ExtentToBack);
			Vis.Shuttle[i].Width    := LREAL_TO_REAL(gShuttleMon.Shuttle[i].Width);
			brsitoa(gShuttleMon.Shuttle[i].Index, ADR(Vis.Shuttle[i].Text));
			Vis.Shuttle[i].ColorRed    := 0.5;    //
			Vis.Shuttle[i].ColorGreen    := 0.5;    // default shuttle color grey
			Vis.Shuttle[i].ColorBlue    := 0.5;        //

			// example: set shuttle colour via user data
			IF gShuttleMon.Shuttle[i].UserData <> 0 THEN
				pUserData ACCESS gShuttleMon.Shuttle[i].UserData;    // access to user data of this shuttle
				IF pUserData.Color = GRAY THEN
					Vis.Shuttle[i].ColorRed    := 0.5;
					Vis.Shuttle[i].ColorGreen    := 0.5;
					Vis.Shuttle[i].ColorBlue    := 0.5;
				ELSIF pUserData.Color = GREEN THEN
					Vis.Shuttle[i].ColorRed    := 0.0;
					Vis.Shuttle[i].ColorGreen    := 1.0;
					Vis.Shuttle[i].ColorBlue    := 0.0;
				ELSIF pUserData.Color = BLUE THEN
					Vis.Shuttle[i].ColorRed    := 0.0;
					Vis.Shuttle[i].ColorGreen    := 0.0;
					Vis.Shuttle[i].ColorBlue    := 1.0;
				ELSIF pUserData.Color = RED THEN
					Vis.Shuttle[i].ColorRed    := 1.0;
					Vis.Shuttle[i].ColorGreen    := 0.0;
					Vis.Shuttle[i].ColorBlue    := 0.0;
				ELSIF pUserData.Color = ORANGE THEN
					Vis.Shuttle[i].ColorRed    := 1.0;
					Vis.Shuttle[i].ColorGreen    := 0.5;
					Vis.Shuttle[i].ColorBlue    := 0.0;
				END_IF
			END_IF

		ELSE
			brsmemset(ADR(Vis.Shuttle[i]), 0, SIZEOF(Vis.Shuttle[0]));
		END_IF

	END_FOR

END_PROGRAM

PROGRAM _EXIT
	(* Insert code here *)

END_PROGRAM
```

### Program Logical/Trak (IEC)

#### Variables.var
```iecst
VAR
	MoveOnSector : BE_MoveOnSector;
	AsmPowerOn : MC_BR_AsmPowerOn_AcpTrak;
	State : USINT;
	AsmReadInfo : MC_BR_AsmReadInfo_AcpTrak;
	AxisArray : ARRAY[1..MAX_SHUTTLES] OF McAxisType;
	FindShuttles : BE_FindShuttles;
END_VAR
```

#### Main.st
```iecst
PROGRAM _INIT
	(* Insert code here *)
	AsmReadInfo.Assembly := ADR(gAssembly_1);
	AsmReadInfo.Enable := TRUE;
	AsmPowerOn.Assembly := ADR(gAssembly_1);
	MoveOnSector.Sector := ADR(Sector_1);
	MoveOnSector.Assembly := ADR(gAssembly_1);
	FindShuttles.Assembly := ADR(gAssembly_1);
END_PROGRAM

PROGRAM _CYCLIC
	CASE State OF
		0://power on
			IF AsmReadInfo.AssemblyInfo.ReadyForPowerOn THEN
				AsmPowerOn.Execute := TRUE;
			END_IF

			IF AsmPowerOn.Done AND AsmReadInfo.AssemblyInfo.PowerOn THEN
				AsmPowerOn.Execute := FALSE;
				State := 1;

			END_IF;

		1: //FIND SHUTTLES
			FindShuttles.Execute := TRUE;
			IF FindShuttles.Done THEN
				FindShuttles.Execute := FALSE;
				AxisArray := FindShuttles.ShuttleAxisArray;
				State := 2;
			END_IF

		2://move shuttles
			MoveOnSector.Acceleration := 10;
			MoveOnSector.Deceleration := 10;
			MoveOnSector.Velocity := 2;
			MoveOnSector.AxisArray := AxisArray;
			MoveOnSector.Execute := TRUE;
			IF MoveOnSector.Done THEN
				MoveOnSector.Execute := FALSE;
				State := 3;
			END_IF

		3: //running

	END_CASE

	AsmReadInfo();
	AsmPowerOn();
	MoveOnSector();
	FindShuttles();

END_PROGRAM

PROGRAM _EXIT
	(* Insert code here *)

END_PROGRAM
```

### Program Logical/SVControl (IEC)

#### Types.typ
```iecst
TYPE
	MoveType_enum :
		(
		LINEAR,
		RADIAL
		);
	Binding_typ : 	STRUCT
		Camera : SceneViewCamera_typ;
		FocalPoint : SceneViewCoord_typ;
		FocalPointVisible : BOOL;
	END_STRUCT;
	Vis_typ : 	STRUCT
		Controls : Controls_typ;
		Bind : Binding_typ;
	END_STRUCT;
	LinearControls_typ : 	STRUCT
		XBtnPos : USINT;
		XBtnNeg : USINT;
		YBtnPos : USINT;
		YBtnNeg : USINT;
		Y : REAL;
		X : REAL;
	END_STRUCT;
	CircularControls_typ : 	STRUCT
		RadiusBtnNeg : USINT;
		RadiusBtnPos : USINT;
		Angle : REAL;
		Radius : REAL;
	END_STRUCT;
	Controls_typ : 	STRUCT
		FocalPoint : FocalPointControls_typ;
		Fov : REAL;
		Z : REAL;
		Circular : CircularControls_typ;
		Linear : LinearControls_typ;
		SavePointA : BOOL;
		MoveType : USINT;
		NewMove : BOOL;
		Start : BOOL;
		Load : BOOL;
		Save : BOOL;
		SelectedMove : USINT;
		MoveMode : MoveType_enum;
	END_STRUCT;
	FocalPointControls_typ : 	STRUCT
		XBtnPos : USINT;
		XBtnNeg : USINT;
		YBtnPos : USINT;
		YBtnNeg : USINT;
		ZBtnPos : USINT;
		ZBtnNeg : USINT;
		Visible : BOOL;
	END_STRUCT;
	Move_typ : 	STRUCT
		IsSaved : BOOL;
		MoveType : MoveType_enum;
		Point : SceneViewCamera_typ;
		FocalPoint : SceneViewCoord_typ;
	END_STRUCT;
	State_enum :
		(
		MOVE_SETTINGS,
		NEW_MOVE,
		UPDATE_LIST,
		NEW_MOVE_SAVE,
		SAVE_MOVE,
		LOAD_MOVE,
		START_MOVE,
		LINEAR_MOVE,
		WAIT_FOR_LINEAR_MOVE_DONE,
		RADIAL_MOVE,
		WAIT_FOR_RADIAL_MOVE_DONE,
		MOVE_COMPLETE,
		WAIT_FOR_STOP
		);
END_TYPE
```

#### Variables.var
```iecst
VAR
	MoveText : STRING[80];
	RadialMove : SV_BE_RadialMove;
	FocalPointMove : SV_BE_FocalPointMove;
	State : State_enum;
	TravelTime : TIME := T#5s;
	Vis : Vis_typ;
	FocalPointInit : SceneViewCoord_typ := (X:=-322,Y:=385,Z:=193);
	StartView : SceneViewCamera_typ := (Perspective:=TRUE,Zoom:=10,Fov:=50,ViewPoint:=(X:=-372,Y:=-861,Z:=840),ViewVector:=(X:=0.05,Y:=0.906,Z:=-0.647),OrientationVector:=(X:=0,Y:=0,Z:=1));
	AngleRad : REAL;
	PointA : SceneViewCamera_typ;
	PointB : SceneViewCamera_typ;
	TotalNumMoves : USINT;
	CompletedMoves : USINT;
	Point : ARRAY[0..2] OF SceneViewCamera_typ;
END_VAR
VAR CONSTANT
	MAX_NUM_MOVES : USINT := 10;
END_VAR
VAR
	MoveNumText : ARRAY[0..MAX_NUM_MOVES] OF STRING[80];
	MoveIndexString : STRING[80];
	IntermediateDateProvider : ARRAY[0..MAX_NUM_MOVES] OF STRING[80];
	DataProvider : ARRAY[0..MAX_NUM_MOVES] OF STRING[80];
	CamMove : ARRAY[0..MAX_NUM_MOVES] OF Move_typ;
	i : USINT;
	FocalPointB : SceneViewCoord_typ;
	FocalPointA : SceneViewCoord_typ;
END_VAR
```

#### Main.st
```iecst
PROGRAM _INIT
	(* Insert code here *)

	Point[0] := StartView;
	Vis.Bind.Camera := StartView;

	Vis.Bind.FocalPoint.X := FocalPointInit.X;
	Vis.Bind.FocalPoint.Y := FocalPointInit.Y;
	Vis.Bind.FocalPoint.Z := FocalPointInit.Z;

	Vis.Controls.Linear.X := StartView.ViewPoint.X;
	Vis.Controls.Linear.Y := StartView.ViewPoint.Y;
	Vis.Controls.Z := StartView.ViewPoint.Z;
	Vis.Controls.Fov := StartView.Fov;
	Vis.Controls.Circular.Radius := 100;
END_PROGRAM

PROGRAM _CYCLIC

	Vis.Bind.FocalPoint.X := Vis.Bind.FocalPoint.X + Vis.Controls.FocalPoint.XBtnPos - Vis.Controls.FocalPoint.XBtnNeg;
	Vis.Bind.FocalPoint.Y := Vis.Bind.FocalPoint.Y + Vis.Controls.FocalPoint.YBtnPos - Vis.Controls.FocalPoint.YBtnNeg;
	Vis.Bind.FocalPoint.Z := Vis.Bind.FocalPoint.Z + Vis.Controls.FocalPoint.ZBtnPos - Vis.Controls.FocalPoint.ZBtnNeg;

	Vis.Controls.Circular.Radius := Vis.Controls.Circular.Radius + Vis.Controls.Circular.RadiusBtnPos - Vis.Controls.Circular.RadiusBtnNeg;
	Vis.Controls.Linear.X := Vis.Controls.Linear.X + Vis.Controls.Linear.XBtnPos - Vis.Controls.Linear.XBtnNeg;
	Vis.Controls.Linear.Y := Vis.Controls.Linear.Y + Vis.Controls.Linear.YBtnPos - Vis.Controls.Linear.YBtnNeg;

	Vis.Bind.FocalPointVisible := Vis.Controls.FocalPoint.Visible;

	CASE State OF
		MOVE_SETTINGS: //set points
			CASE Vis.Controls.MoveMode OF
				LINEAR:
					MoveText := 'Linear';
					Vis.Bind.Camera.ViewPoint.X := Vis.Controls.Linear.X;
					Vis.Bind.Camera.ViewPoint.Y := Vis.Controls.Linear.Y;

					AngleRad := atan2((Vis.Bind.Camera.ViewPoint.Y - Vis.Bind.FocalPoint.Y),(Vis.Bind.Camera.ViewPoint.X - Vis.Bind.FocalPoint.X));
					Vis.Controls.Circular.Angle := AngleRad * 180 / PI;
					IF Vis.Controls.Circular.Angle < 0 THEN
						Vis.Controls.Circular.Angle := Vis.Controls.Circular.Angle + 360;
					ELSIF Vis.Controls.Circular.Angle >= 360 THEN
						Vis.Controls.Circular.Angle := Vis.Controls.Circular.Angle - 360;
					END_IF
					Vis.Controls.Circular.Radius := (Vis.Bind.Camera.ViewPoint.X - Vis.Bind.FocalPoint.X) / COS(AngleRad);
				RADIAL:
					MoveText := 'Radial';
					AngleRad := Vis.Controls.Circular.Angle * PI / 180;

					Vis.Bind.Camera.ViewPoint.X := (Vis.Controls.Circular.Radius * COS(AngleRad)) + Vis.Bind.FocalPoint.X;
					Vis.Bind.Camera.ViewPoint.Y := (Vis.Controls.Circular.Radius * SIN(AngleRad)) + Vis.Bind.FocalPoint.Y;

					Vis.Controls.Linear.X := Vis.Bind.Camera.ViewPoint.X;
					Vis.Controls.Linear.Y := Vis.Bind.Camera.ViewPoint.Y;
			END_CASE

			Vis.Bind.Camera.OrientationVector.X := 0;
			Vis.Bind.Camera.OrientationVector.Y := 0;
			Vis.Bind.Camera.OrientationVector.Z := 1;

			Vis.Bind.Camera.ViewPoint.Z := Vis.Controls.Z;
			Vis.Bind.Camera.Fov := Vis.Controls.Fov;

			Vis.Bind.Camera.ViewVector.X := (Vis.Bind.FocalPoint.X - Vis.Bind.Camera.ViewPoint.X) / 1000.0;
			Vis.Bind.Camera.ViewVector.Y := (Vis.Bind.FocalPoint.Y - Vis.Bind.Camera.ViewPoint.Y) / 1000.0;
			Vis.Bind.Camera.ViewVector.Z := (Vis.Bind.FocalPoint.Z - Vis.Bind.Camera.ViewPoint.Z) / 1000.0;

			IF Vis.Controls.NewMove THEN
				Vis.Controls.NewMove := FALSE;
				State := NEW_MOVE;
			ELSIF Vis.Controls.Load THEN
				State := LOAD_MOVE;
			ELSIF Vis.Controls.Save THEN
				Vis.Controls.Save := FALSE;
				State := SAVE_MOVE;
			END_IF

			IF Vis.Controls.SavePointA THEN
				Vis.Controls.SavePointA := FALSE;
				Point[0] := Vis.Bind.Camera;
			END_IF

			IF Vis.Controls.Start THEN
				CompletedMoves := 0;
				PointA := Point[0];
				PointB := CamMove[0].Point;
				FocalPointA := FocalPointInit;
				FocalPointB := CamMove[0].FocalPoint;
				State := START_MOVE;
			END_IF

		NEW_MOVE: //new move
			FOR i := 0 TO MAX_NUM_MOVES DO
				IF NOT CamMove[i].IsSaved THEN
					CamMove[i].IsSaved := TRUE;
					CamMove[i].MoveType := Vis.Controls.MoveMode;

					State := UPDATE_LIST;
					EXIT;
				ELSIF i = MAX_NUM_MOVES THEN
					State := MOVE_SETTINGS;
				END_IF
			END_FOR

		UPDATE_LIST:
			brsftoa(i, ADR(MoveIndexString));
			MoveNumText[i] := CONCAT(MoveIndexString, ': ');
			MoveNumText[i] := CONCAT(MoveNumText[i], MoveText);
			MoveNumText[i] := CONCAT(MoveNumText[i], ' Move');

			IntermediateDateProvider[i] := CONCAT('{"value":"',MoveIndexString);
			IntermediateDateProvider[i] := CONCAT(IntermediateDateProvider[i],'","text":"');
			IntermediateDateProvider[i] := CONCAT(IntermediateDateProvider[i], MoveNumText[i]);
			DataProvider[i] := CONCAT(IntermediateDateProvider[i],'"}');

			State := NEW_MOVE_SAVE;

		NEW_MOVE_SAVE:

			TotalNumMoves := TotalNumMoves + 1;
			CamMove[i].Point := Vis.Bind.Camera;
			CamMove[i].FocalPoint := Vis.Bind.FocalPoint;
			State := MOVE_SETTINGS;

		LOAD_MOVE: //load
			Vis.Controls.Load := FALSE;

			IF CamMove[Vis.Controls.SelectedMove].IsSaved THEN
				Vis.Controls.Linear.X := CamMove[Vis.Controls.SelectedMove].Point.ViewPoint.X;
				Vis.Controls.Linear.Y := CamMove[Vis.Controls.SelectedMove].Point.ViewPoint.Y;
				Vis.Controls.Z := CamMove[Vis.Controls.SelectedMove].Point.ViewPoint.Z;
				Vis.Controls.Fov := CamMove[Vis.Controls.SelectedMove].Point.Fov;

				Vis.Bind.Camera := CamMove[Vis.Controls.SelectedMove].Point;
				Vis.Bind.FocalPoint := CamMove[Vis.Controls.SelectedMove].FocalPoint;
			END_IF
			State := MOVE_SETTINGS;

		SAVE_MOVE: //save
			IF CamMove[Vis.Controls.SelectedMove].IsSaved THEN
				CamMove[Vis.Controls.SelectedMove].Point := Vis.Bind.Camera;
				CamMove[Vis.Controls.SelectedMove].FocalPoint := Vis.Bind.FocalPoint;
			END_IF
			State := MOVE_SETTINGS;

		START_MOVE:
			IF CamMove[CompletedMoves].MoveType = LINEAR THEN
				State := LINEAR_MOVE;
			ELSIF CamMove[CompletedMoves].MoveType = RADIAL THEN
				State := RADIAL_MOVE;
			END_IF

		RADIAL_MOVE:
			Vis.Controls.SelectedMove := CompletedMoves;
			RadialMove.PointA := PointA;
			RadialMove.PointB := PointB;
			RadialMove.FocalPointA := FocalPointA;
			RadialMove.FocalPointB := FocalPointB;
			RadialMove.TravelTime := TravelTime;
			RadialMove.Execute := TRUE;
			State := WAIT_FOR_RADIAL_MOVE_DONE;

//			IF RadialMove.Done THEN
//				RadialMove.Execute := FALSE;
//				CompletedMoves := CompletedMoves + 1;
//				State := MOVE_COMPLETE;
//			END_IF

		WAIT_FOR_RADIAL_MOVE_DONE:

			IF RadialMove.Done THEN
				RadialMove.Execute := FALSE;
				CompletedMoves := CompletedMoves + 1;
				State := MOVE_COMPLETE;
			END_IF

			RadialMove();
			Vis.Bind.FocalPoint := RadialMove.FocalPointPos;
			Vis.Bind.Camera := RadialMove.SceneViewPos;

		LINEAR_MOVE:
			Vis.Controls.SelectedMove := CompletedMoves;
			FocalPointMove.PointA := PointA;
			FocalPointMove.PointB := PointB;
			//FocalPointMove.FocalPoint := Vis.FocalPoint;
			FocalPointMove.FocalPointA := FocalPointA;
			FocalPointMove.FocalPointB := FocalPointB;
			FocalPointMove.TravelTime := TravelTime;
			FocalPointMove.Execute := TRUE;
			State := WAIT_FOR_LINEAR_MOVE_DONE;

		WAIT_FOR_LINEAR_MOVE_DONE:

			IF FocalPointMove.Done THEN
				FocalPointMove.Execute := FALSE;
				CompletedMoves := CompletedMoves + 1;
				State := MOVE_COMPLETE;
			END_IF

			FocalPointMove();
			Vis.Bind.FocalPoint := FocalPointMove.FocalPointPos;
			Vis.Bind.Camera := FocalPointMove.SceneViewPos;

		MOVE_COMPLETE:
			IF CompletedMoves < TotalNumMoves THEN
				PointA := Vis.Bind.Camera;
				PointB := CamMove[CompletedMoves].Point;
				FocalPointA := Vis.Bind.FocalPoint;
				FocalPointB := CamMove[CompletedMoves].FocalPoint;
				State := START_MOVE;
			ELSE
				State := WAIT_FOR_STOP;
			END_IF

		WAIT_FOR_STOP:
			IF NOT Vis.Controls.Start THEN
				State := MOVE_SETTINGS;
			END_IF

	END_CASE

//	RadialMove();
//	FocalPointMove();

END_PROGRAM

PROGRAM _EXIT
	(* Insert code here *)

END_PROGRAM
```

- Visualisation Logical/mappView (not shown)

Listed in the project but not available here: Logical/Global.typ, Logical/Global.var
